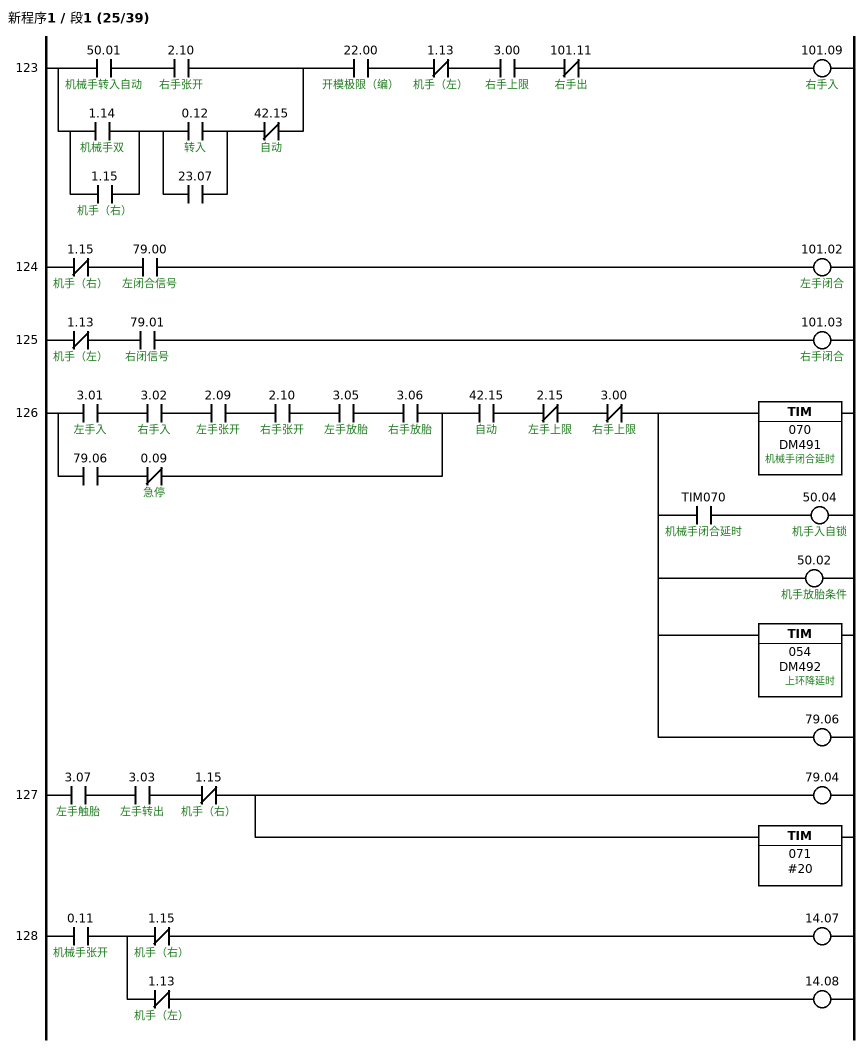
; [picture p24: 新程序1 / 段1, rungs 123-128]
; rung 123
LD 50.01  ; 机械手转入自动
AND 2.10  ; 右手张开
LD 1.14  ; 机械手双
OR 1.15  ; 机手（右）
LD 0.12  ; 转入
OR 23.07
ANDLD
ANDNOT 42.15  ; 自动
ORLD
AND 22.00  ; 开模极限（编）
ANDNOT 1.13  ; 机手（左）
AND 3.00  ; 右手上限
ANDNOT 101.11  ; 右手出
OUT 101.09  ; 右手入
; rung 124
LDNOT 1.15  ; 机手（右）
AND 79.00  ; 左闭合信号
OUT 101.02  ; 左手闭合
; rung 125
LDNOT 1.13  ; 机手（左）
AND 79.01  ; 右闭信号
OUT 101.03  ; 右手闭合
; rung 126
LD 3.01  ; 左手入
AND 3.02  ; 右手入
AND 2.09  ; 左手张开
AND 2.10  ; 右手张开
AND 3.05  ; 左手放胎
AND 3.06  ; 右手放胎
LD 79.06
ANDNOT 0.09  ; 急停
ORLD
AND 42.15  ; 自动
ANDNOT 2.15  ; 左手上限
ANDNOT 3.00  ; 右手上限
OUT TR0
TIM 070 DM491  ; 机械手闭合延时
AND TIM070  ; 机械手闭合延时
OUT 50.04  ; 机手入自锁
LD TR0
OUT 50.02  ; 机手放胎条件
TIM 054 DM492  ; 上环降延时
OUT 79.06
; rung 127
LD 3.07  ; 左手触胎
AND 3.03  ; 左手转出
ANDNOT 1.15  ; 机手（右）
OUT 79.04
TIM 071 #20
; rung 128
LD 0.11  ; 机械手张开
OUT TR0
ANDNOT 1.15  ; 机手（右）
OUT 14.07
LD TR0
ANDNOT 1.13  ; 机手（左）
OUT 14.08

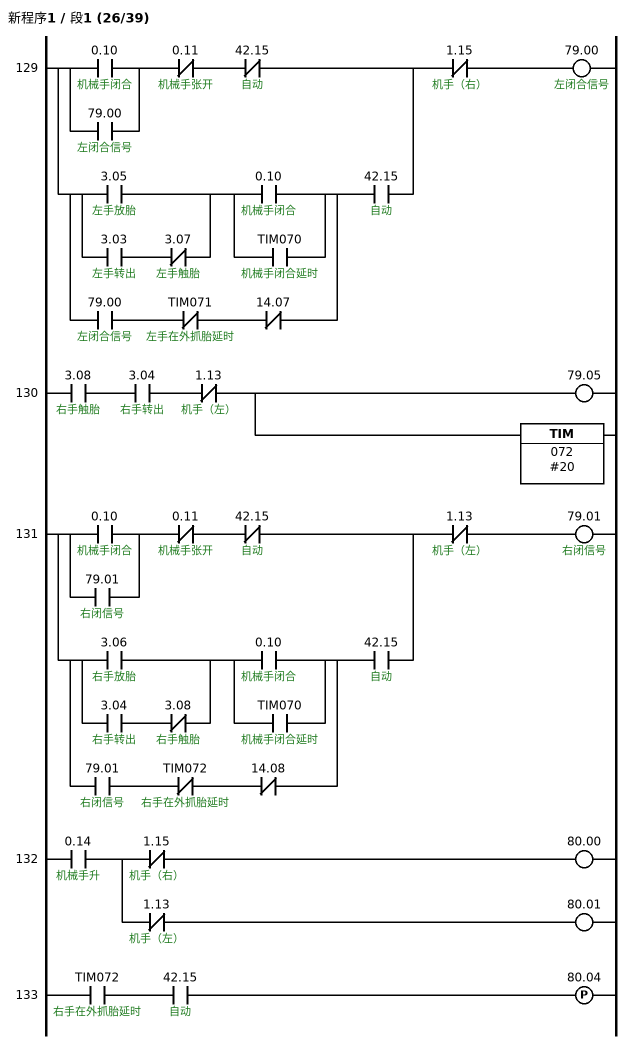
; rung 129
LD 0.10  ; 机械手闭合
OR 79.00  ; 左闭合信号
ANDNOT 0.11  ; 机械手张开
ANDNOT 42.15  ; 自动
LD 3.05  ; 左手放胎
LD 3.03  ; 左手转出
ANDNOT 3.07  ; 左手触胎
ORLD
LD 0.10  ; 机械手闭合
OR TIM070  ; 机械手闭合延时
ANDLD
LD 79.00  ; 左闭合信号
ANDNOT TIM071  ; 左手在外抓胎延时
ANDNOT 14.07
ORLD
AND 42.15  ; 自动
ORLD
ANDNOT 1.15  ; 机手（右）
OUT 79.00  ; 左闭合信号
; rung 130
LD 3.08  ; 右手触胎
AND 3.04  ; 右手转出
ANDNOT 1.13  ; 机手（左）
OUT 79.05
TIM 072 #20
; rung 131
LD 0.10  ; 机械手闭合
OR 79.01  ; 右闭信号
ANDNOT 0.11  ; 机械手张开
ANDNOT 42.15  ; 自动
LD 3.06  ; 右手放胎
LD 3.04  ; 右手转出
ANDNOT 3.08  ; 右手触胎
ORLD
LD 0.10  ; 机械手闭合
OR TIM070  ; 机械手闭合延时
ANDLD
LD 79.01  ; 右闭信号
ANDNOT TIM072  ; 右手在外抓胎延时
ANDNOT 14.08
ORLD
AND 42.15  ; 自动
ORLD
ANDNOT 1.13  ; 机手（左）
OUT 79.01  ; 右闭信号
; rung 132
LD 0.14  ; 机械手升
OUT TR0
ANDNOT 1.15  ; 机手（右）
OUT 80.00
LD TR0
ANDNOT 1.13  ; 机手（左）
OUT 80.01
; rung 133
LD TIM072  ; 右手在外抓胎延时
AND 42.15  ; 自动
DIFU(13) 80.04

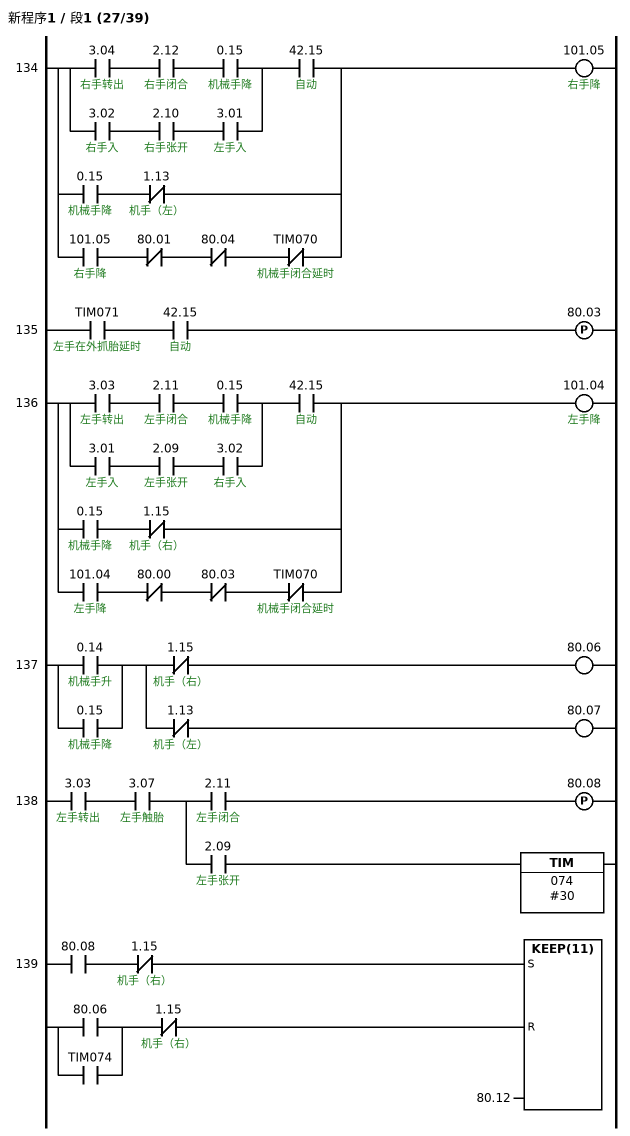
; rung 134
LD 3.04  ; 右手转出
AND 2.12  ; 右手闭合
AND 0.15  ; 机械手降
LD 3.02  ; 右手入
AND 2.10  ; 右手张开
AND 3.01  ; 左手入
ORLD
AND 42.15  ; 自动
LD 0.15  ; 机械手降
ANDNOT 1.13  ; 机手（左）
ORLD
LD 101.05  ; 右手降
ANDNOT 80.01
ANDNOT 80.04
ANDNOT TIM070  ; 机械手闭合延时
ORLD
OUT 101.05  ; 右手降
; rung 135
LD TIM071  ; 左手在外抓胎延时
AND 42.15  ; 自动
DIFU(13) 80.03
; rung 136
LD 3.03  ; 左手转出
AND 2.11  ; 左手闭合
AND 0.15  ; 机械手降
LD 3.01  ; 左手入
AND 2.09  ; 左手张开
AND 3.02  ; 右手入
ORLD
AND 42.15  ; 自动
LD 0.15  ; 机械手降
ANDNOT 1.15  ; 机手（右）
ORLD
LD 101.04  ; 左手降
ANDNOT 80.00
ANDNOT 80.03
ANDNOT TIM070  ; 机械手闭合延时
ORLD
OUT 101.04  ; 左手降
; rung 137
LD 0.14  ; 机械手升
OR 0.15  ; 机械手降
OUT TR0
ANDNOT 1.15  ; 机手（右）
OUT 80.06
LD TR0
ANDNOT 1.13  ; 机手（左）
OUT 80.07
; rung 138
LD 3.03  ; 左手转出
AND 3.07  ; 左手触胎
OUT TR0
AND 2.11  ; 左手闭合
DIFU(13) 80.08
LD TR0
AND 2.09  ; 左手张开
TIM 074 #30
; rung 139
LD 80.08
ANDNOT 1.15  ; 机手（右）
LD 80.06
OR TIM074
ANDNOT 1.15  ; 机手（右）
KEEP(11) 80.12

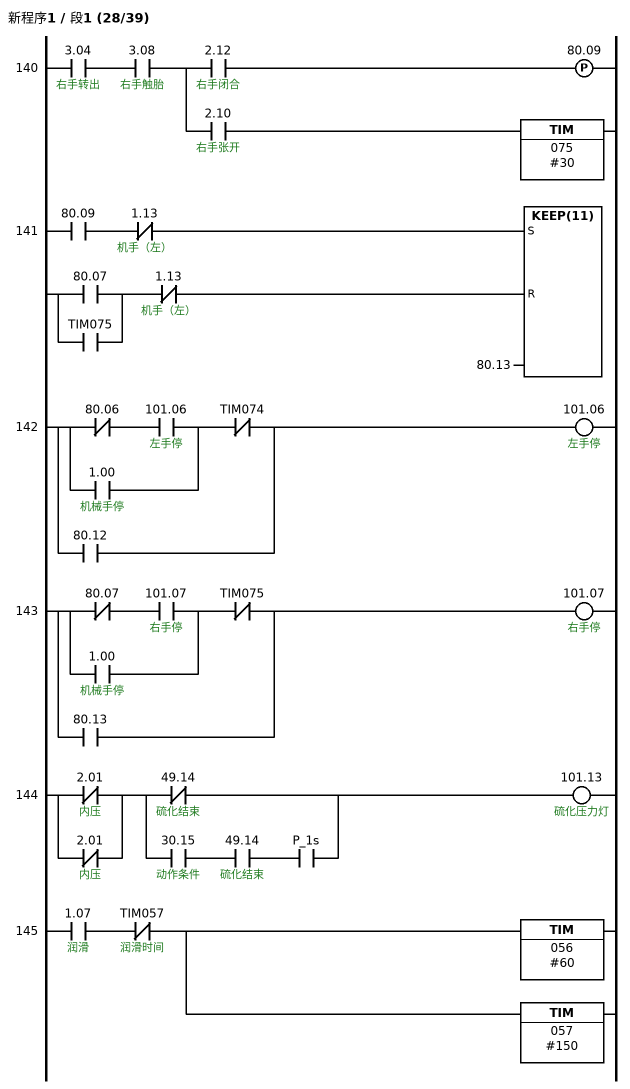
; rung 140
LD 3.04  ; 右手转出
AND 3.08  ; 右手触胎
OUT TR0
AND 2.12  ; 右手闭合
DIFU(13) 80.09
LD TR0
AND 2.10  ; 右手张开
TIM 075 #30
; rung 141
LD 80.09
ANDNOT 1.13  ; 机手（左）
LD 80.07
OR TIM075
ANDNOT 1.13  ; 机手（左）
KEEP(11) 80.13
; rung 142
LDNOT 80.06
AND 101.06  ; 左手停
OR 1.00  ; 机械手停
ANDNOT TIM074
OR 80.12
OUT 101.06  ; 左手停
; rung 143
LDNOT 80.07
AND 101.07  ; 右手停
OR 1.00  ; 机械手停
ANDNOT TIM075
OR 80.13
OUT 101.07  ; 右手停
; rung 144
LDNOT 2.01  ; 内压
ORNOT 2.01  ; 内压
LDNOT 49.14  ; 硫化结束
LD 30.15  ; 动作条件
AND 49.14  ; 硫化结束
AND P_1s
ORLD
ANDLD
OUT 101.13  ; 硫化压力灯
; rung 145
LD 1.07  ; 润滑
ANDNOT TIM057  ; 润滑时间
TIM 056 #60
TIM 057 #150

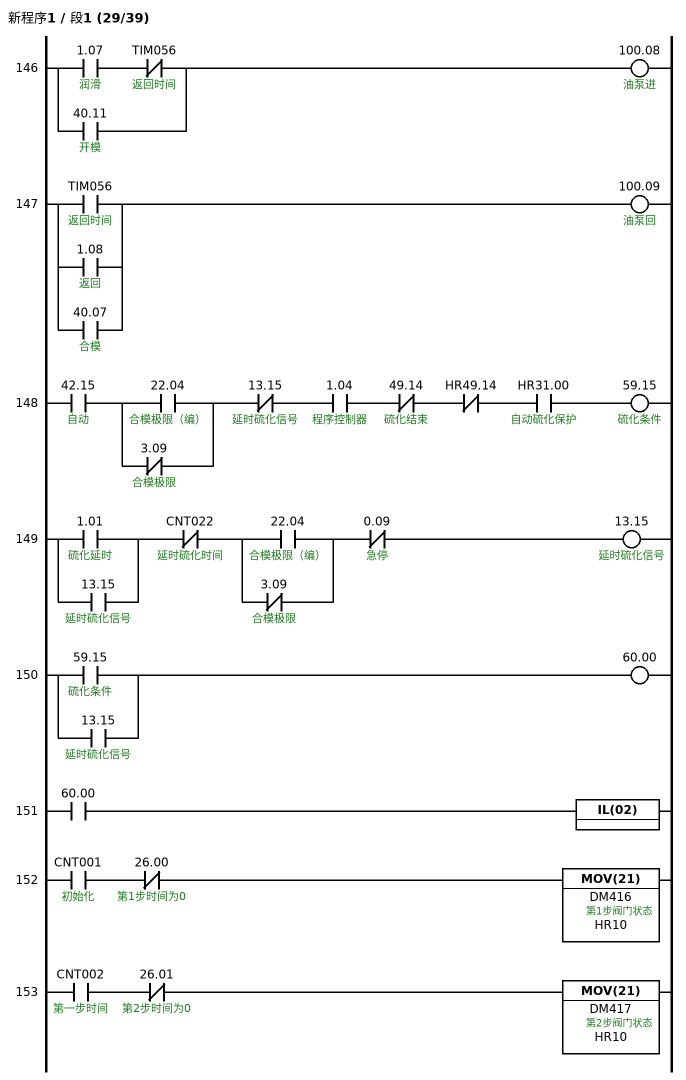
; rung 146
LD 1.07  ; 润滑
ANDNOT TIM056  ; 返回时间
OR 40.11  ; 开模
OUT 100.08  ; 油泵进
; rung 147
LD TIM056  ; 返回时间
OR 1.08  ; 返回
OR 40.07  ; 合模
OUT 100.09  ; 油泵回
; rung 148
LD 42.15  ; 自动
LD 22.04  ; 合模极限（编）
ORNOT 3.09  ; 合模极限
ANDLD
ANDNOT 13.15  ; 延时硫化信号
AND 1.04  ; 程序控制器
ANDNOT 49.14  ; 硫化结束
ANDNOT HR49.14
AND HR31.00  ; 自动硫化保护
OUT 59.15  ; 硫化条件
; rung 149
LD 1.01  ; 硫化延时
OR 13.15  ; 延时硫化信号
ANDNOT CNT022  ; 延时硫化时间
LD 22.04  ; 合模极限（编）
ORNOT 3.09  ; 合模极限
ANDLD
ANDNOT 0.09  ; 急停
OUT 13.15  ; 延时硫化信号
; rung 150
LD 59.15  ; 硫化条件
OR 13.15  ; 延时硫化信号
OUT 60.00
; rung 151
LD 60.00
IL(02)
; rung 152
LD CNT001  ; 初始化
ANDNOT 26.00  ; 第1步时间为0
MOV(21) DM416 HR10  ; 第1步阀门状态
; rung 153
LD CNT002  ; 第一步时间
ANDNOT 26.01  ; 第2步时间为0
MOV(21) DM417 HR10  ; 第2步阀门状态

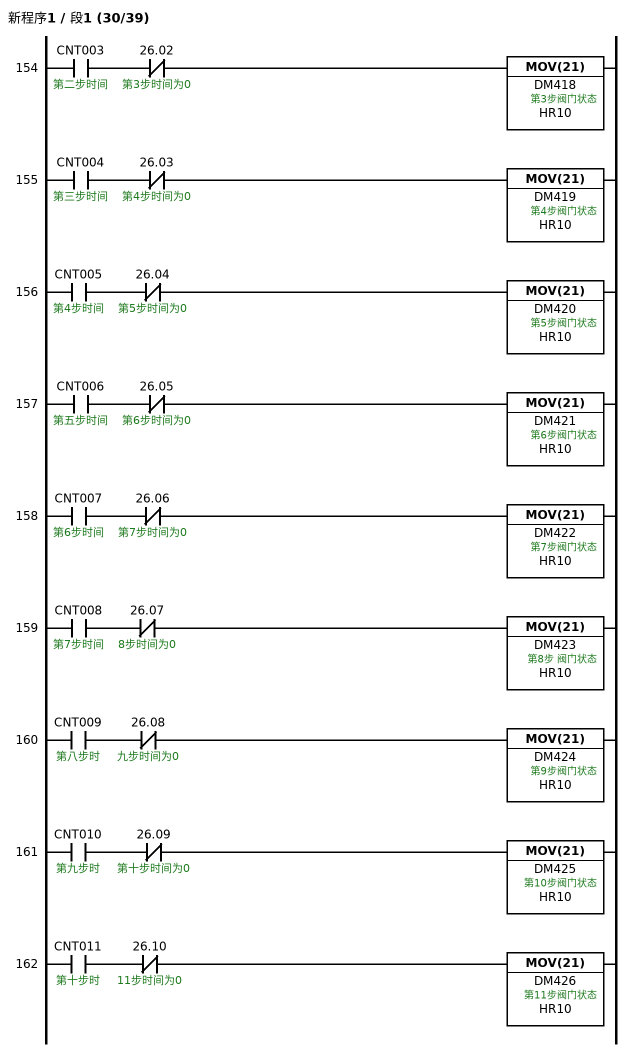
; rung 154
LD CNT003  ; 第二步时间
ANDNOT 26.02  ; 第3步时间为0
MOV(21) DM418 HR10  ; 第3步阀门状态
; rung 155
LD CNT004  ; 第三步时间
ANDNOT 26.03  ; 第4步时间为0
MOV(21) DM419 HR10  ; 第4步阀门状态
; rung 156
LD CNT005  ; 第4步时间
ANDNOT 26.04  ; 第5步时间为0
MOV(21) DM420 HR10  ; 第5步阀门状态
; rung 157
LD CNT006  ; 第五步时间
ANDNOT 26.05  ; 第6步时间为0
MOV(21) DM421 HR10  ; 第6步阀门状态
; rung 158
LD CNT007  ; 第6步时间
ANDNOT 26.06  ; 第7步时间为0
MOV(21) DM422 HR10  ; 第7步阀门状态
; rung 159
LD CNT008  ; 第7步时间
ANDNOT 26.07  ; 8步时间为0
MOV(21) DM423 HR10  ; 第8步 阀门状态
; rung 160
LD CNT009  ; 第八步时
ANDNOT 26.08  ; 九步时间为0
MOV(21) DM424 HR10  ; 第9步阀门状态
; rung 161
LD CNT010  ; 第九步时
ANDNOT 26.09  ; 第十步时间为0
MOV(21) DM425 HR10  ; 第10步阀门状态
; rung 162
LD CNT011  ; 第十步时
ANDNOT 26.10  ; 11步时间为0
MOV(21) DM426 HR10  ; 第11步阀门状态

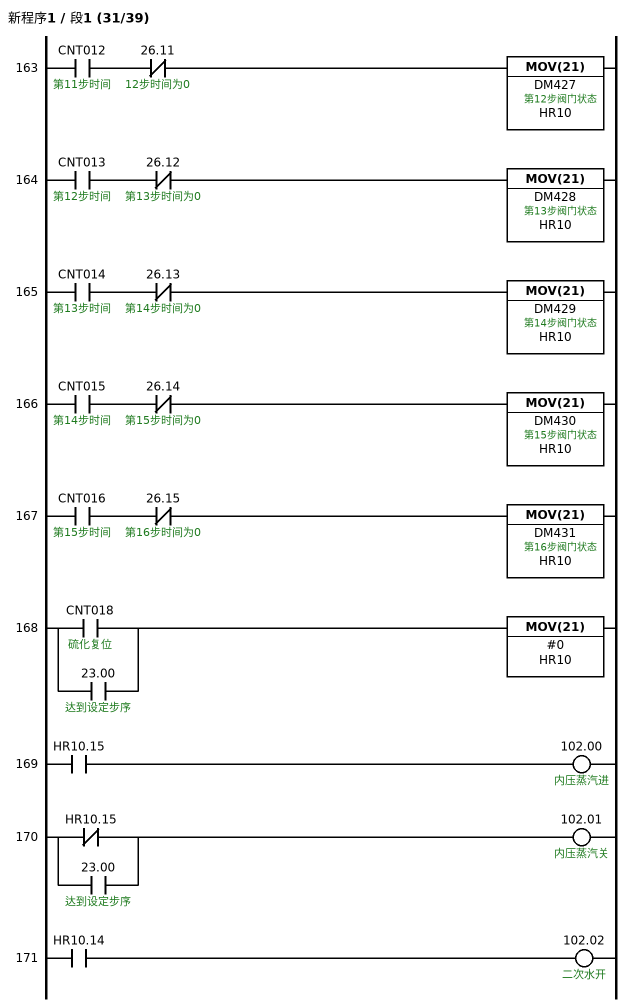
; rung 163
LD CNT012  ; 第11步时间
ANDNOT 26.11  ; 12步时间为0
MOV(21) DM427 HR10  ; 第12步阀门状态
; rung 164
LD CNT013  ; 第12步时间
ANDNOT 26.12  ; 第13步时间为0
MOV(21) DM428 HR10  ; 第13步阀门状态
; rung 165
LD CNT014  ; 第13步时间
ANDNOT 26.13  ; 第14步时间为0
MOV(21) DM429 HR10  ; 第14步阀门状态
; rung 166
LD CNT015  ; 第14步时间
ANDNOT 26.14  ; 第15步时间为0
MOV(21) DM430 HR10  ; 第15步阀门状态
; rung 167
LD CNT016  ; 第15步时间
ANDNOT 26.15  ; 第16步时间为0
MOV(21) DM431 HR10  ; 第16步阀门状态
; rung 168
LD CNT018  ; 硫化复位
OR 23.00  ; 达到设定步序
MOV(21) #0 HR10
; rung 169
LD HR10.15
OUT 102.00  ; 内压蒸汽进
; rung 170
LDNOT HR10.15
OR 23.00  ; 达到设定步序
OUT 102.01  ; 内压蒸汽关
; rung 171
LD HR10.14
OUT 102.02  ; 二次水开

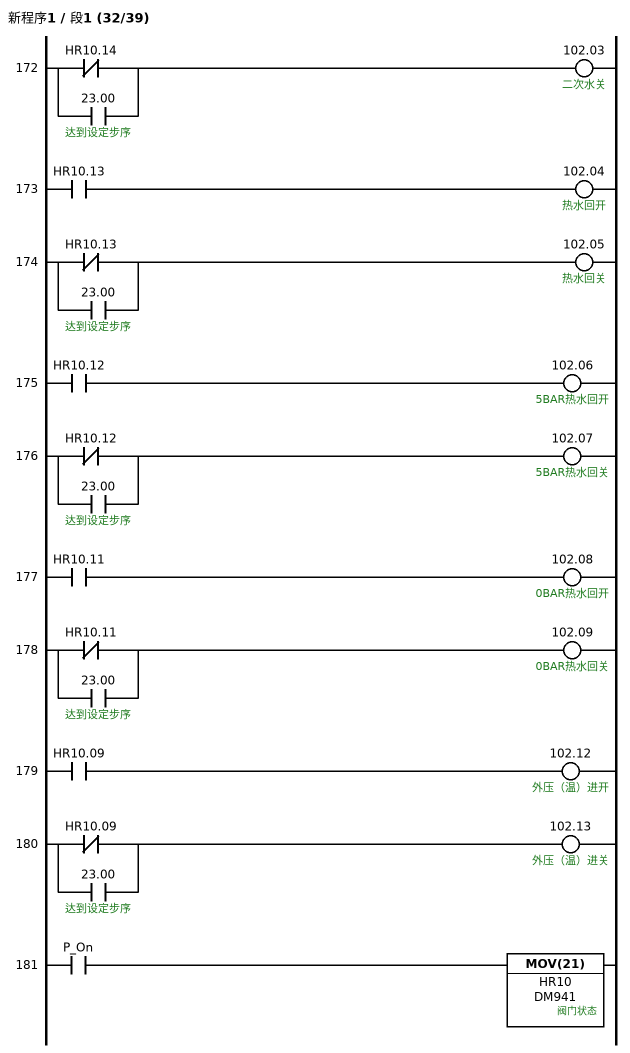
; rung 172
LDNOT HR10.14
OR 23.00  ; 达到设定步序
OUT 102.03  ; 二次水关
; rung 173
LD HR10.13
OUT 102.04  ; 热水回开
; rung 174
LDNOT HR10.13
OR 23.00  ; 达到设定步序
OUT 102.05  ; 热水回关
; rung 175
LD HR10.12
OUT 102.06  ; 5BAR热水回开
; rung 176
LDNOT HR10.12
OR 23.00  ; 达到设定步序
OUT 102.07  ; 5BAR热水回关
; rung 177
LD HR10.11
OUT 102.08  ; 0BAR热水回开
; rung 178
LDNOT HR10.11
OR 23.00  ; 达到设定步序
OUT 102.09  ; 0BAR热水回关
; rung 179
LD HR10.09
OUT 102.12  ; 外压（温）进开
; rung 180
LDNOT HR10.09
OR 23.00  ; 达到设定步序
OUT 102.13  ; 外压（温）进关
; rung 181
LD P_On
MOV(21) HR10 DM941  ; 阀门状态

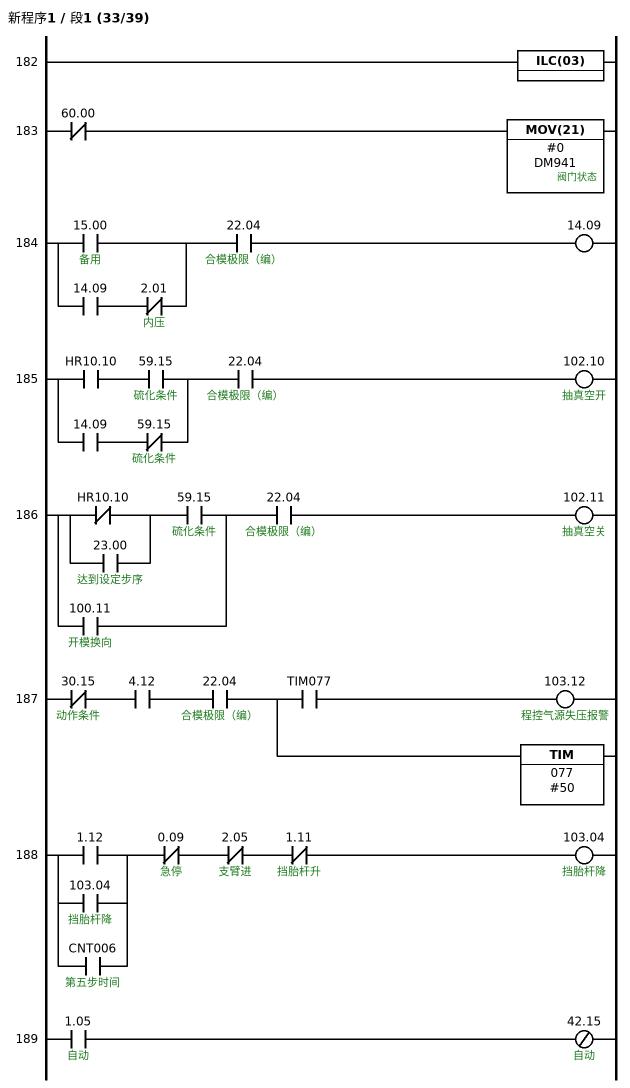
; rung 182
ILC(03)
; rung 183
LDNOT 60.00
MOV(21) #0 DM941  ; 阀门状态
; rung 184
LD 15.00  ; 备用
LD 14.09
ANDNOT 2.01  ; 内压
ORLD
AND 22.04  ; 合模极限（编）
OUT 14.09
; rung 185
LD HR10.10
AND 59.15  ; 硫化条件
LD 14.09
ANDNOT 59.15  ; 硫化条件
ORLD
AND 22.04  ; 合模极限（编）
OUT 102.10  ; 抽真空开
; rung 186
LDNOT HR10.10
OR 23.00  ; 达到设定步序
AND 59.15  ; 硫化条件
OR 100.11  ; 开模换向
AND 22.04  ; 合模极限（编）
OUT 102.11  ; 抽真空关
; rung 187
LDNOT 30.15  ; 动作条件
AND 4.12
AND 22.04  ; 合模极限（编）
OUT TR0
AND TIM077
OUT 103.12  ; 程控气源失压报警
LD TR0
TIM 077 #50
; rung 188
LD 1.12
OR 103.04  ; 挡胎杆降
OR CNT006  ; 第五步时间
ANDNOT 0.09  ; 急停
ANDNOT 2.05  ; 支臂进
ANDNOT 1.11  ; 挡胎杆升
OUT 103.04  ; 挡胎杆降
; rung 189
LD 1.05  ; 自动
OUTNOT 42.15  ; 自动

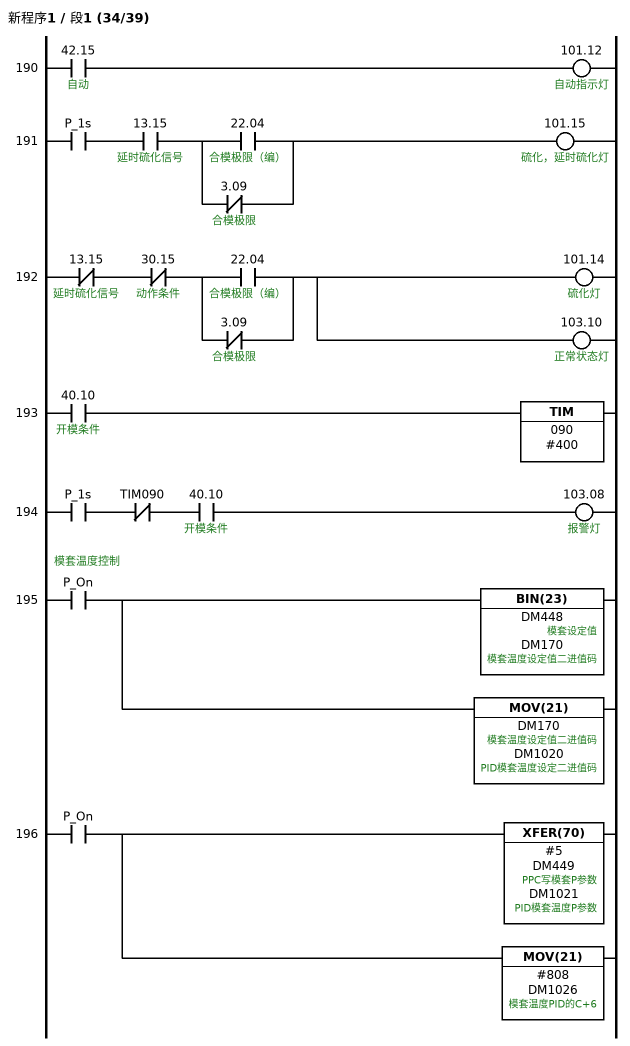
; rung 190
LD 42.15  ; 自动
OUT 101.12  ; 自动指示灯
; rung 191
LD P_1s
AND 13.15  ; 延时硫化信号
LD 22.04  ; 合模极限（编）
ORNOT 3.09  ; 合模极限
ANDLD
OUT 101.15  ; 硫化，延时硫化灯
; rung 192
LDNOT 13.15  ; 延时硫化信号
ANDNOT 30.15  ; 动作条件
LD 22.04  ; 合模极限（编）
ORNOT 3.09  ; 合模极限
ANDLD
OUT 101.14  ; 硫化灯
OUT 103.10  ; 正常状态灯
; rung 193
LD 40.10  ; 开模条件
TIM 090 #400
; rung 194
LD P_1s
ANDNOT TIM090
AND 40.10  ; 开模条件
OUT 103.08  ; 报警灯
; rung 195: 模套温度控制
LD P_On
BIN(23) DM448 DM170  ; 模套设定值, 模套温度设定值二进值码
MOV(21) DM170 DM1020  ; 模套温度设定值二进值码, PID模套温度设定二进值码
; rung 196
LD P_On
XFER(70) #5 DM449 DM1021  ; PPC写模套P参数, PID模套温度P参数
MOV(21) #808 DM1026  ; 模套温度PID的C+6

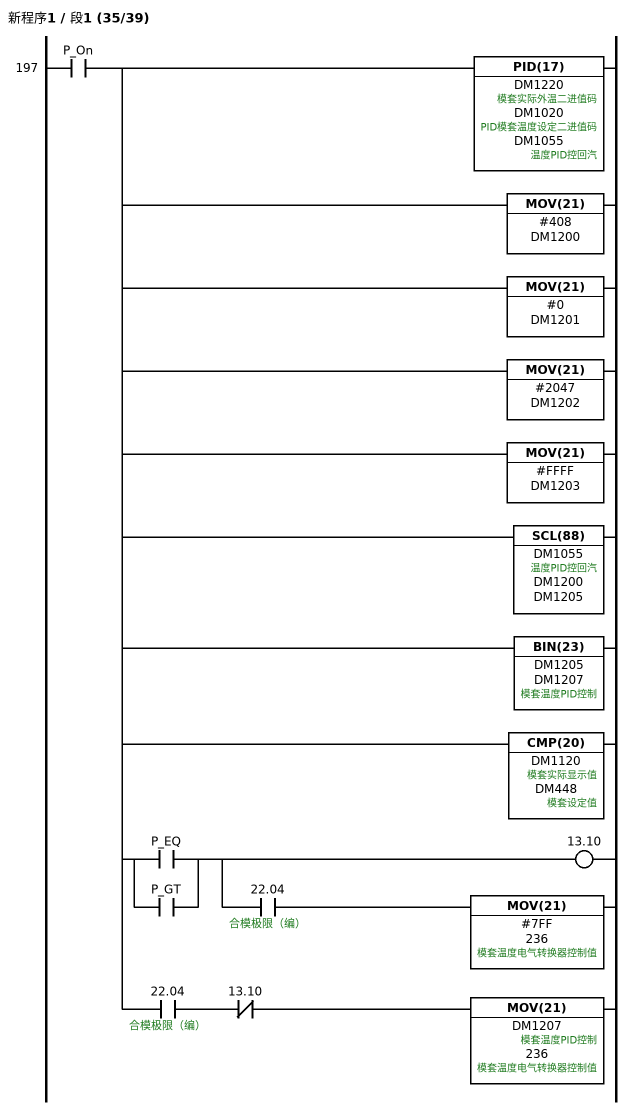
; rung 197
LD P_On
OUT TR0
PID(17) DM1220 DM1020 DM1055  ; 模套实际外温二进值码, PID模套温度设定二进值码, 温度PID控回汽
MOV(21) #408 DM1200
MOV(21) #0 DM1201
MOV(21) #2047 DM1202
MOV(21) #FFFF DM1203
SCL(88) DM1055 DM1200 DM1205  ; 温度PID控回汽
BIN(23) DM1205 DM1207  ; 模套温度PID控制
CMP(20) DM1120 DM448  ; 模套实际显示值, 模套设定值
LD P_EQ
OR P_GT
ANDLD
OUT 13.10
AND 22.04  ; 合模极限（编）
MOV(21) #7FF 236  ; 模套温度电气转换器控制值
LD TR0
AND 22.04  ; 合模极限（编）
ANDNOT 13.10
MOV(21) DM1207 236  ; 模套温度PID控制, 模套温度电气转换器控制值

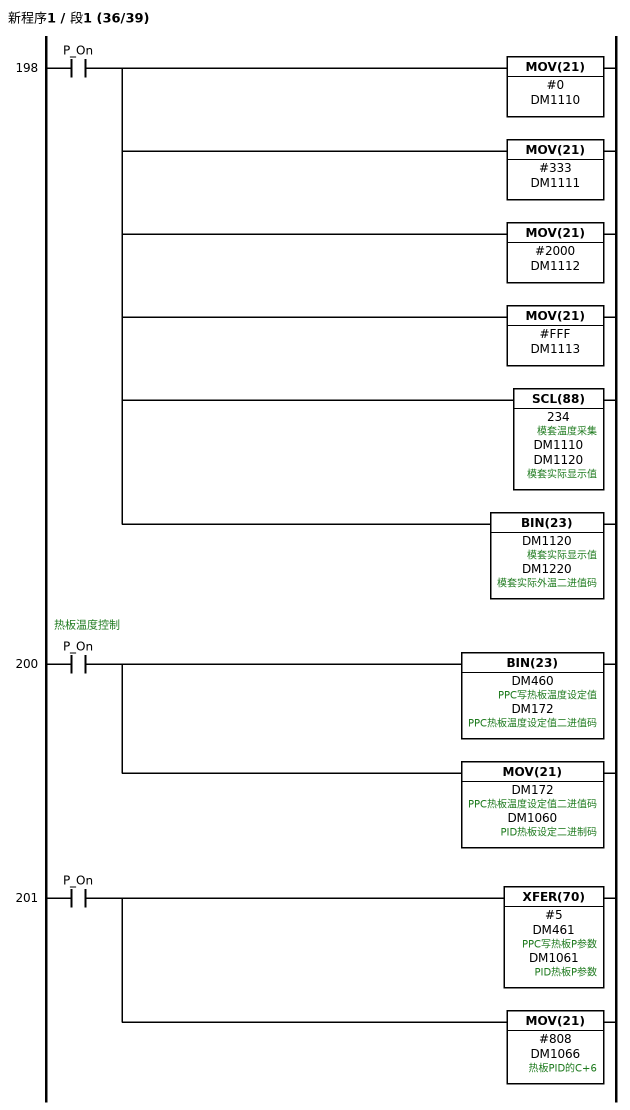
; rung 198
LD P_On
MOV(21) #0 DM1110
MOV(21) #333 DM1111
MOV(21) #2000 DM1112
MOV(21) #FFF DM1113
SCL(88) 234 DM1110 DM1120  ; 模套温度采集, 模套实际显示值
BIN(23) DM1120 DM1220  ; 模套实际显示值, 模套实际外温二进值码
; rung 200: 热板温度控制
LD P_On
BIN(23) DM460 DM172  ; PPC写热板温度设定值, PPC热板温度设定值二进值码
MOV(21) DM172 DM1060  ; PPC热板温度设定值二进值码, PID热板设定二进制码
; rung 201
LD P_On
XFER(70) #5 DM461 DM1061  ; PPC写热板P参数, PID热板P参数
MOV(21) #808 DM1066  ; 热板PID的C+6

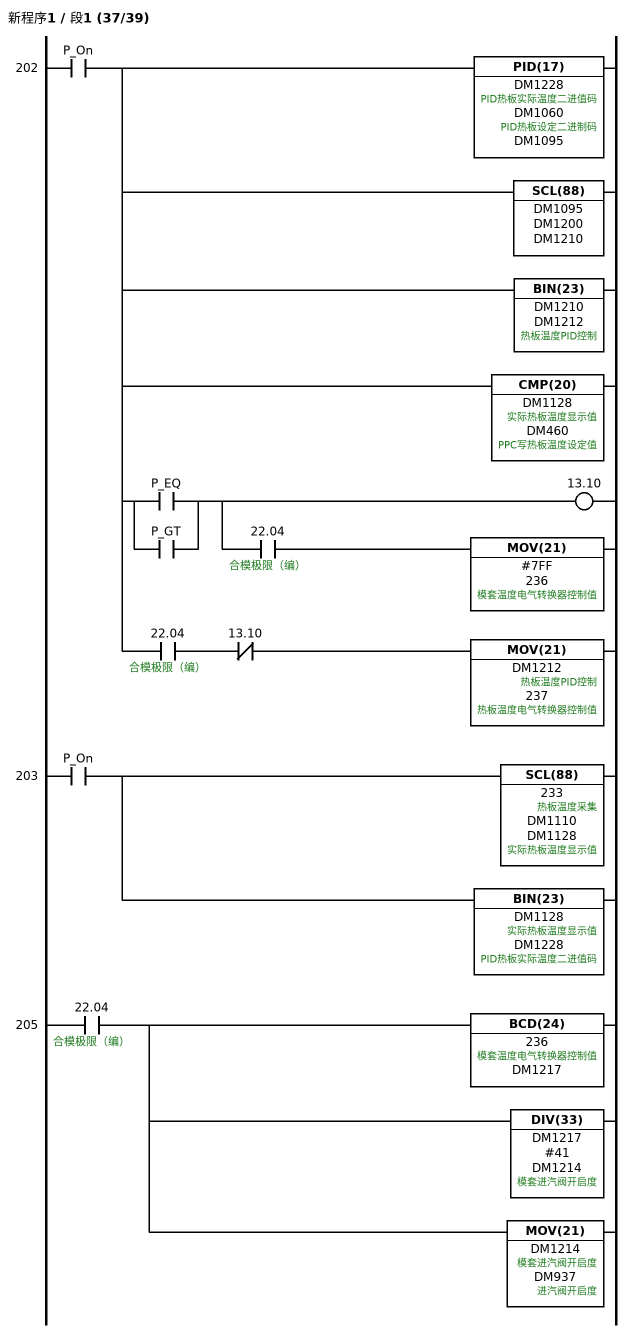
; rung 202
LD P_On
OUT TR0
PID(17) DM1228 DM1060 DM1095  ; PID热板实际温度二进值码, PID热板设定二进制码
SCL(88) DM1095 DM1200 DM1210
BIN(23) DM1210 DM1212  ; 热板温度PID控制
CMP(20) DM1128 DM460  ; 实际热板温度显示值, PPC写热板温度设定值
LD P_EQ
OR P_GT
ANDLD
OUT 13.10
AND 22.04  ; 合模极限（编）
MOV(21) #7FF 236  ; 模套温度电气转换器控制值
LD TR0
AND 22.04  ; 合模极限（编）
ANDNOT 13.10
MOV(21) DM1212 237  ; 热板温度PID控制, 热板温度电气转换器控制值
; rung 203
LD P_On
SCL(88) 233 DM1110 DM1128  ; 热板温度采集, 实际热板温度显示值
BIN(23) DM1128 DM1228  ; 实际热板温度显示值, PID热板实际温度二进值码
; rung 205
LD 22.04  ; 合模极限（编）
BCD(24) 236 DM1217  ; 模套温度电气转换器控制值
DIV(33) DM1217 #41 DM1214  ; 模套进汽阀开启度
MOV(21) DM1214 DM937  ; 模套进汽阀开启度, 进汽阀开启度

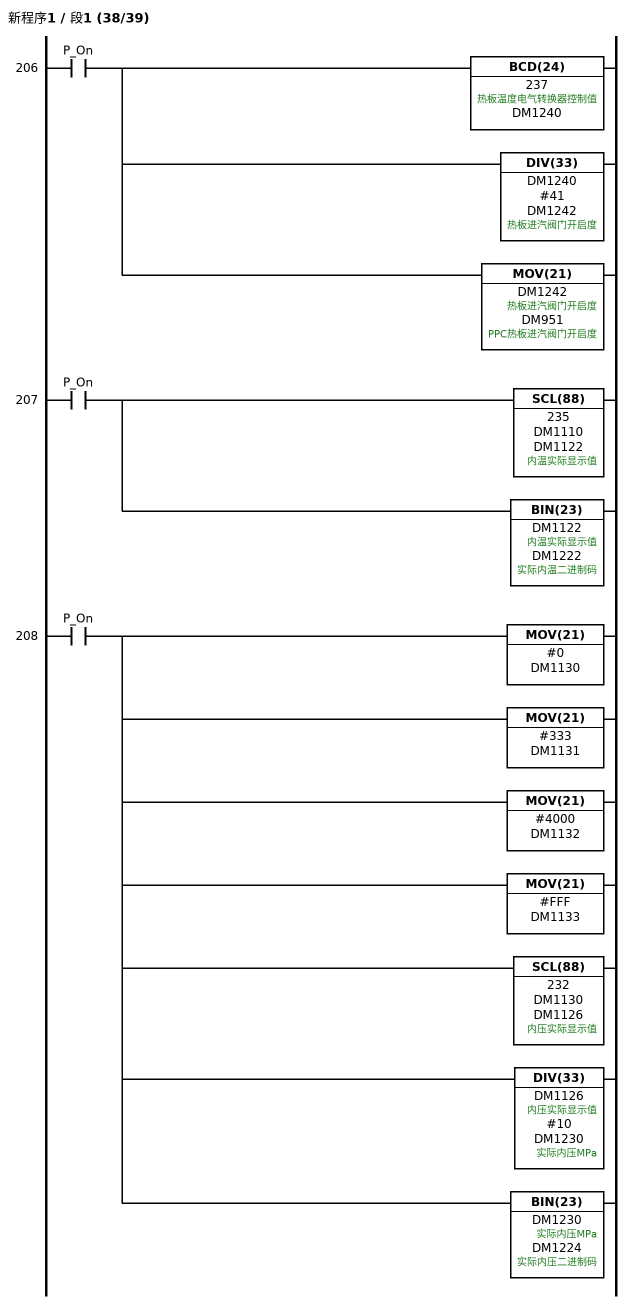
; rung 206
LD P_On
BCD(24) 237 DM1240  ; 热板温度电气转换器控制值
DIV(33) DM1240 #41 DM1242  ; 热板进汽阀门开启度
MOV(21) DM1242 DM951  ; 热板进汽阀门开启度, PPC热板进汽阀门开启度
; rung 207
LD P_On
SCL(88) 235 DM1110 DM1122  ; 内温实际显示值
BIN(23) DM1122 DM1222  ; 内温实际显示值, 实际内温二进制码
; rung 208
LD P_On
MOV(21) #0 DM1130
MOV(21) #333 DM1131
MOV(21) #4000 DM1132
MOV(21) #FFF DM1133
SCL(88) 232 DM1130 DM1126  ; 内压实际显示值
DIV(33) DM1126 #10 DM1230  ; 内压实际显示值, 实际内压MPa
BIN(23) DM1230 DM1224  ; 实际内压MPa, 实际内压二进制码

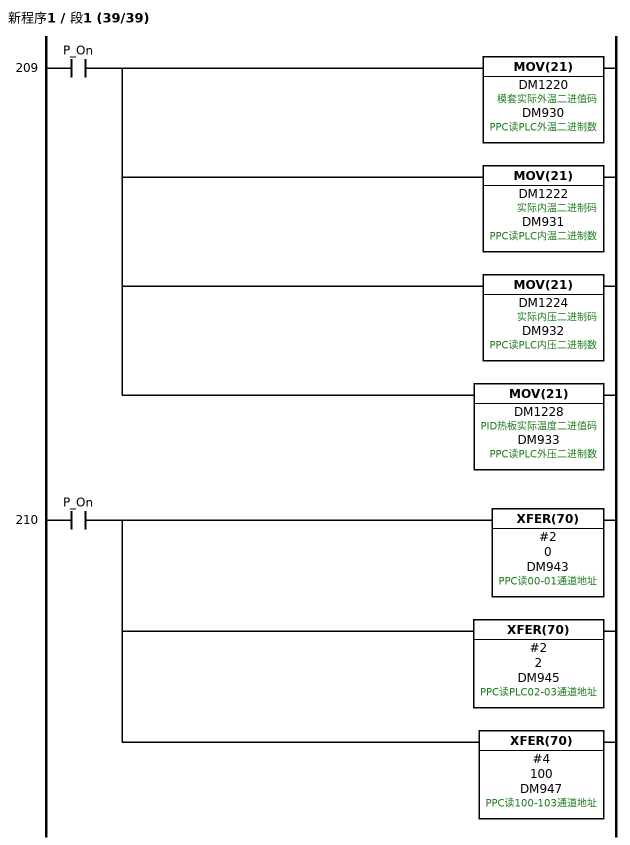
; rung 209
LD P_On
MOV(21) DM1220 DM930  ; 模套实际外温二进值码, PPC读PLC外温二进制数
MOV(21) DM1222 DM931  ; 实际内温二进制码, PPC读PLC内温二进制数
MOV(21) DM1224 DM932  ; 实际内压二进制码, PPC读PLC内压二进制数
MOV(21) DM1228 DM933  ; PID热板实际温度二进值码, PPC读PLC外压二进制数
; rung 210
LD P_On
XFER(70) #2 0 DM943  ; PPC读00-01通道地址
XFER(70) #2 2 DM945  ; PPC读PLC02-03通道地址
XFER(70) #4 100 DM947  ; PPC读100-103通道地址
; rung 211
END(01)